RoboDK station: welding.rdk

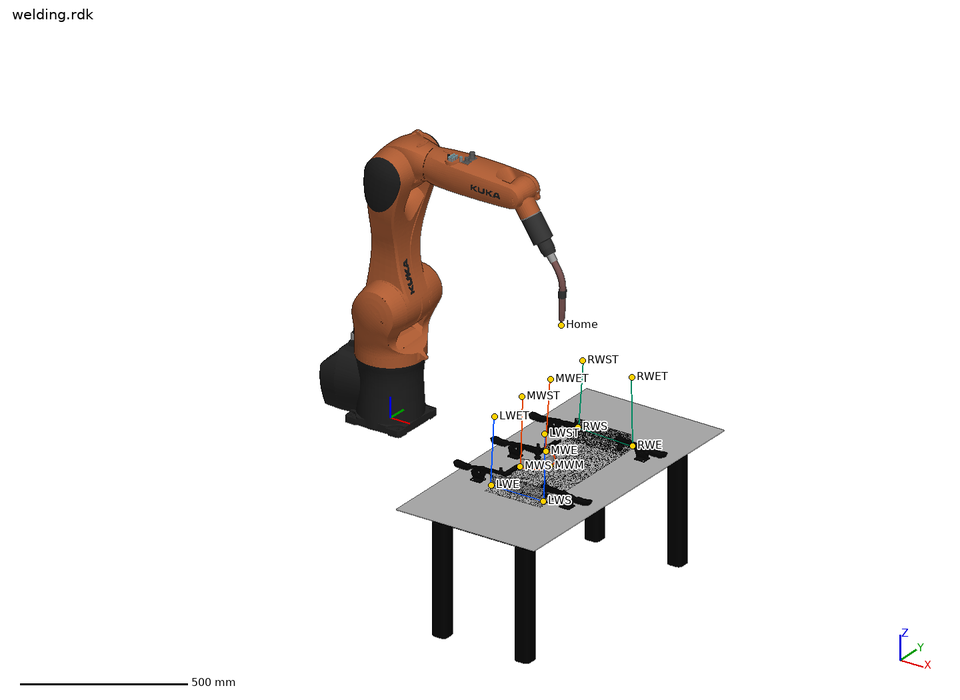
[picture v0: the station drawn from its stored meshes, robots at their saved joint values, targets as dots, program paths as lines]
Station Welding (saved by RoboDK 5.8.0). Poses are relative to the parent item; angles as X-Y-Z fixed-axis rotations.
  - frame KUKA KR 10 R900 sixx Base at (-17.95, 0, 0) mm
    - robot KUKA KR 10 R900 sixx: 6 axes, payload 10 kg, reach 901 mm, repeatability 0.03 mm, weight 52 kg
        modified DH rows (alpha deg, a mm, theta deg, d mm): 0, 0, 0, 400; -90, 25, 0, 0; 0, 455, -90, 0; -90, 35, 0, 420; 90, 0, 0, 0; -90, 0, 180, 80
        joint limits [-170, -190, -120, -185, -120, -350] to [170, 45, 156, 185, 120, 350]; home [0, -90, 90, 0, 0, 0]; saved at [0, -87.202, 88.365, 0, 55.85, 0]
      - tool Generic Welding Gun (Through-arm), TCP at (89, 0, 340) mm, rotated rx 0 ry 35 rz 0 deg, size 122.1 x 64 x 340.8 mm
    - object Weld-1 at (369.21, -499, 0) mm, rotated rx 0 ry 0 rz 90.34 deg, size 1000 x 500 x 492.1 mm, geometry from Weld-1.stl
    - target Home (Cartesian target) at (621.85, 0, 480.18) mm, rotated rx -180 ry -2.01 rz -180 deg; joints [0, -87.202, 88.365, 0, 55.85, 0] of KUKA KR 10 R900 sixx
    - target MWS (Cartesian target) at (517.26, -63.96, 8.14) mm, rotated rx 132.44 ry -2.01 rz 180 deg; joints [44.743, -38.507, 116.157, -79.359, 56.465, 101.039] of KUKA KR 10 R900 sixx
    - target MWM (Cartesian target) at (585.08, -5.13, 5.17) mm, rotated rx -179.13 ry -48.94 rz 179.37 deg; joints [0.09, -29.469, 67.715, -179.363, -65.698, 179.708] of KUKA KR 10 R900 sixx
    - target MWE (Cartesian target) at (518.69, 67.6, 6.71) mm, rotated rx -136.07 ry -2.01 rz 180 deg; joints [-43.444, -40.981, 118.002, 80.907, 53.381, -102.736] of KUKA KR 10 R900 sixx
    - target LWE (Cartesian target) at (527.54, -230.56, 14.32) mm, rotated rx 144.9 ry 0.15 rz 180 deg; joints [51.917, -41.24, 105.422, 112.344, -53.488, -83.461] of KUKA KR 10 R900 sixx
    - target LWS (Cartesian target) at (718.75, -230.56, 14.81) mm, rotated rx 144.9 ry 0.15 rz 180 deg; joints [39.774, -30.888, 80.26, 114.227, -53.189, -103.653] of KUKA KR 10 R900 sixx
    - target LWET (Cartesian target) at (538.52, -228.7, 245.27) mm, rotated rx -180 ry -2.01 rz 180 deg; joints [30.744, -83.117, 117.094, -32.667, 31.04, 55.298] of KUKA KR 10 R900 sixx
    - target LWST (Cartesian target) at (721.76, -228.7, 238.83) mm, rotated rx -180 ry -2.01 rz 180 deg; joints [21.941, -63.805, 92.162, -22.208, 32.561, 37.657] of KUKA KR 10 R900 sixx
    - target RWST (Cartesian target) at (534.09, 237.3, 245.43) mm, rotated rx 180 ry -2.01 rz -180 deg; joints [-31.979, -83.045, 116.986, 33.357, 31.628, -56.913] of KUKA KR 10 R900 sixx
    - target RWET (Cartesian target) at (712.91, 237.3, 239.14) mm, rotated rx 180 ry -2.01 rz -180 deg; joints [-23.006, -64.384, 92.994, 23.202, 32.69, -39.44] of KUKA KR 10 R900 sixx
    - target RWE (Cartesian target) at (716.7, 237.3, 11.17) mm, rotated rx -133.19 ry -2.01 rz -180 deg; joints [-43.259, -21.204, 67.103, 63.365, 65.635, -66.703] of KUKA KR 10 R900 sixx
    - target RWS (Cartesian target) at (517.31, 237.3, 18.18) mm, rotated rx -133.19 ry -2.01 rz -180 deg; joints [-55.66, -32.99, 94.741, 61.334, 64.804, -85.853] of KUKA KR 10 R900 sixx
    - target MWET (Cartesian target) at (528.78, 77.18, 245.62) mm, rotated rx -180 ry -2.01 rz 180 deg; joints [-11.637, -91.084, 125.506, 15.709, 23.93, -24.219] of KUKA KR 10 R900 sixx
    - target MWST (Cartesian target) at (528.78, -69.78, 245.62) mm, rotated rx -180 ry -2.01 rz 180 deg; joints [10.547, -91.265, 125.683, -14.355, 23.701, 22.065] of KUKA KR 10 R900 sixx
  - program reset (1 instructions, listed below)
  - program weldleft (8 instructions, listed below)
  - Python program WeldOn (listed below)
  - program weldmiddle (8 instructions, listed below)
  - program weldright (8 instructions, listed below)
  - program main (8 instructions, listed below)
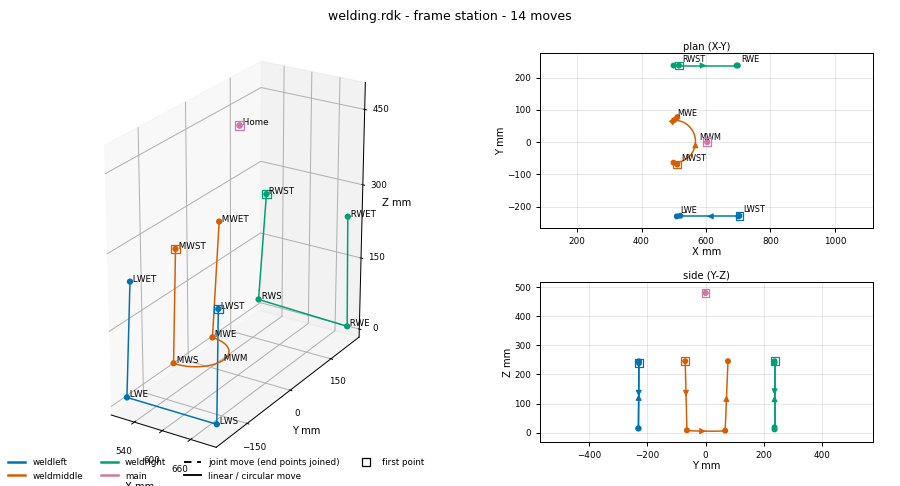
[picture p0: tool path of welding.rdk in frame station, 14 of 14 moves have a stored position in this frame; points joined in program order, loops and branches not executed]

--- program reset (robot KUKA KR 10 R900 sixx) ---
  Replace objects

--- program weldleft (robot KUKA KR 10 R900 sixx) ---
  Set Ref.: KUKA KR 10 R900 sixx Base
  Set Tool: Generic Welding Gun (Through-arm)
  MoveJ (LWST)
  MoveL (LWS)
  Call WeldOn(1)
  MoveL (LWE)
  Call WeldOn(0)
  MoveL (LWET)

--- Python program WeldOn ---
# This macro allows simulating the material deposition of a weld gun
# By default, this macro will activate the trace once it is called.
# Run the macro ArcEnd to stop the trace.
#
# The macros ArcStart, ArcEnd and WeldOn, SpindleOn, all behave in a similar way, the only difference is the default behavior
# This behavior simmulates Fanuc Arc Welding and triggers appropriate output when using the customized post processor.
# Select ESC to clear the trace manually.
#
# It is possible to call WeldOn(ON) to simulate turning the material deposition ON or WeldOn(OFF) to stop simulating the gun
# Calling WeldOn(RESET) clears all displayed data.
# The macro will output spray gun statistics
#
# Optional:
#     This macro can manage multiple guns and multiple colors.
#     As an example, you can call this macro the following way:
#
# WeldOn(State, ToolName, Color)
#     State: [ON/OFF/RESET]
#     TorchName: The name of the tool. For example: Tool 1
#     Color: A named color or a hex color in the format: '#AARRGGBB'
#             Important: for full color definition you should provide Alpha channel first
#
# Examples:
#     WeldOn(ON)                 # Turn on the trace using the default color
#     WeldOn(OFF)                # Turn off the tool trace
#     WeldOn(ON, Tool 1, yellow) # Turn on the trace for tool 1 in yellow
#     WeldOn(ON, Tool 2, blue) # Turn on the trace for tool 2 in blue
#     WeldOn(OFF, Torch1)        # Turn off trace for Torch 1
#     WeldOn(ON, Torch1, #889900FF) # Turn on the trace for torch 2 in a violet color
#     WeldOn(ON, ,red)         # Turn on the trace for a generic torch in red color
#
# --------------------------------------------------------------
# This script shows how to create "spray" object in RoboDK that allows simulating particle deposition by using:
# RDK.Spray_Add(tool, object, options_command, volume, geometry)
#    tool: tool item (TCP) to use
#    object: object to project the particles
#    options_command (optional): string to specify options.
#    volume (optional): Matrix of parameters defining the volume of the spray gun
#    geometry (optional): Matrix of vertices defining the triangles.
#
# More information here:
# https://robodk.com/doc/en/PythonAPI/robodk.html#robodk.robolink.Robolink.Spray_Add
# https://robodk.com/doc/en/RoboDK-API.html
#
# The scripts ArcStart, ArcEnd and WeldOn and SpindleOn behave in a similar way, the only difference is the default behavior
# This behavior simmulates Fanuc Arc Welding and triggers appropriate output when using the customized post processor.
# Select ESC to clear the trace manually.
#
# Example scripts that use Spray_Add:
#     SpindleOn / SpindleOff    -> Turn trace On/Off
#     ArcOn / ArcOff            -> Turn trace On/Off
#     SprayOn / SprayOff        -> Simulate a spray given a workspace volume (for painting)
#     WeldOn / WeldOff          -> Support for multiple weld guns
#
#----------------------------------------------------------

# Constant variables for the first parameter:
ACTION_RESET = -1  # Same as: RESET (clear all traces)
ACTION_OFF = 0  # Same as: OFF (turn on)
ACTION_ON = 1  # Same as: ON (turn off)

# Define the default Action (ACTION_OFF to deactivate, ACTION_ON to activate, ACTION_RESET to clear any spray gun/trace)
# Setting it to None will display a message
Action = ACTION_ON

# Define the default color as a named color or as #AARRGGBB (Alpha, Red, Green Blue)
# COLOR = 'blue'
COLOR = '#CC3344FF'  # AARRGGBB

# Use a specific tool as a spray gun
Tool_Name = None  # Use the active tool
#Tool_Name = 'Torch1'

# Use a specific object to project particles:
Object_Name = None  # Use the first object in the active reference frame
#Object_Name = 'Part'

# --------------------------------------------------
# Program start:
from robodk.robolink import *  # API to communicate with RoboDK
from robodk.robodialogs import *

RDK = Robolink()

# quit if we are not in simulation mode
if RDK.RunMode() != RUNMODE_SIMULATE:
    quit()

# Check command input (parameters passed in the call). This is the same as if we were doing a command line call passing parameters.
import sys
if len(sys.argv) > 1:
    Action_str = sys.argv[1].strip().upper()
    if 'ON' in Action_str:
        Action = ACTION_ON
    elif 'OFF' in Action_str:
        Action = ACTION_OFF
    elif 'RESET' in Action_str:
        Action = ACTION_RESET
    else:
        Action = int(Action_str)

    if len(sys.argv) > 2:
        Tool_Name = sys.argv[2].strip()
        if Tool_Name == '':
            Tool_Name = None

        if len(sys.argv) > 3:
            COLOR = sys.argv[3].lower().strip()

# Display summary
print("Applying action: " + str(Action))
print("Using tool: " + str(Tool_Name))
print("Using color: " + COLOR)

# Get any previously added spray gun simulations and display statistics (spray on the part vs spray falling out of the part)
info, data = RDK.Spray_GetStats()
n_sprays = data.size(1)
spray_id = -1
if n_sprays > 0 and Tool_Name is not None:
    spray_id = RDK.getParam(Tool_Name)
    if spray_id is None or Action == ACTION_ON or type(spray_id) == str or spray_id >= n_sprays:
        spray_id = -1

    print("Spray gun statistics:")
    print(info)
    print(data.tr())
    # # Diplay statistics
    # RDK.ShowMessage("Material used: %.1f%%<br>Material waisted: %.1f%%<br>Total particles: %.1f" % (data[1,0],data[2,0],data[3,0]), True)
    # # Clear previous spray
    # RDK.Spray_Clear()

# If the default Action is None, display a message to activate/deactivate the spray gun
if Action is None:
    print('Note: This macro can be called as ArcStart(1) or ArcStart(0) or ArcStart(-1)')
    entry = mbox('Turn gun ON or OFF', ('On', '1'), ('Off', '0'))
    if not entry:
        quit()
    Action = int(entry)

# Apply the desired action
if Action == ACTION_OFF:
    # Turn the gun off
    RDK.Spray_SetState(SPRAY_OFF, spray_id)

elif Action == ACTION_OFF:
    # Clear all spray simulations (same as pressing ESC key)
    RDK.Spray_Clear(spray_id)

elif Action == ACTION_ON:
    # Create a new spray gun object in RoboDK
    # by using RDK.Spray_Add(tool, object, options_command, volume, geometry)
    # tool: tool item (TCP) to use
    # object: object to project the particles
    # options_command (optional): string to specify options. Example:
    #     STEP=AxB: Defines the grid to be projected 1x1 means only one line of particle projection (for example, for welding)
    #     PARTICLE: Defines the shape and size of particle (sphere or particle), unless a specific geometry is provided:
    #       a- SPHERE(radius, facets)
    #       b- SPHERE(radius, facets, scalex, scaley, scalez)
    #       b- CUBE(sizex, sizey, sizez)
    #     RAND=factor: Defines a random factor factor 0 means that the particles are not deposited randomly
    #     ELLYPSE: defines the volume as an ellypse (default)
    #     RECTANGLE: defines the volume as a rectangle
    #     PROJECT: project the particles to the surface (default) (for welding, painting or scanning)
    #     NO_PROJECT: does not project the particles to the surface (for example, for 3D printing)
    #
    # volume (optional): Matrix of parameters defining the volume of the spray gun
    # geometry (optional): Matrix of vertices defining the triangles.

    if spray_id < 0:
        tool = 0  # auto detect active tool
        obj = 0  # auto detect object in active reference frame
        if Tool_Name is not None:
            tool = RDK.Item(Tool_Name, ITEM_TYPE_TOOL)

        if Object_Name is not None:
            obj = RDK.Item(Object_Name, ITEM_TYPE_OBJECT)
        # We can specify a given tool object and/or object
        #robot = RDK.Item("ABB IRB 2600-12/1.85", ITEM_TYPE_ROBOT)
        #tools = robot.Childs()
        #if len(tools) > 0:
        #    tool = tools[0]
        #obj = RDK.Item('object', ITEM_TYPE_OBJECT)

        # Create volume parameters
        options_command = "NO_PROJECT PARTICLE=SPHERE(2,8,1,1,1) STEP=1x0 RAND=0 COLOR=" + COLOR

        spray_id = RDK.Spray_Add(tool, obj, options_command)

    # Remember the ID of the spray gun for later
    if Tool_Name is not None:
        RDK.setParam(Tool_Name, spray_id)

    # Apply the state to activate the trace
    RDK.Spray_SetState(SPRAY_ON, spray_id)

--- program weldmiddle (robot KUKA KR 10 R900 sixx) ---
  Set Ref.: KUKA KR 10 R900 sixx Base
  Set Tool: Generic Welding Gun (Through-arm)
  MoveJ (MWST)
  MoveL (MWS)
  Call WeldOn(1)
  MoveC (MWM, MWE)
  Call WeldOn(0)
  MoveL (MWET)

--- program weldright (robot KUKA KR 10 R900 sixx) ---
  Set Ref.: KUKA KR 10 R900 sixx Base
  Set Tool: Generic Welding Gun (Through-arm)
  MoveJ (RWST)
  MoveL (RWS)
  Call WeldOn(1)
  MoveL (RWE)
  Call WeldOn(0)
  MoveL (RWET)

--- program main (robot KUKA KR 10 R900 sixx) ---
  Set Ref.: KUKA KR 10 R900 sixx Base
  Set Tool: Generic Welding Gun (Through-arm)
  MoveJ (Home)
  Call weldleft
  Call weldmiddle
  Call weldright
  Call reset
  MoveJ (Home)
